{attribute 'qualified_only'}
VAR_GLOBAL
	HMIStartStatusLamp : BOOL := FALSE;
	HMIStopStatusLamp : BOOL := FALSE;
	HMIErrorStatusLamp : BOOL := FALSE;
	
	HMIStartMachine : BOOL := FALSE;
	HMIStopMachine : BOOL := FALSE;
END_VAR

(* stored: Version 1.1.0.1
   GVL HMIInterface: Id {4d023906-a51a-4956-9ce5-a29a374d340f} *)
